PROGRAM MAIN
VAR
	previousTime: ULINT := 0;
	currentTime: ULINT := 0;
	
	loTime: ULINT := 0;
	hiTime: ULINT := 0;
	getTime: GETSYSTEMTIME;
	
	deltaTime: REAL := 0.0;
	
	skogestadPID: Skogestad;
	parallelPID: ParallelPID;

	
	lastPID: REAL := 0;
	useSkogestad: BOOL := TRUE;
	
	init: BOOL := TRUE;
END_VAR

IF init THEN
	lastPID := GVL.kp + GVL.ki + GVL.kd;
	init := FALSE;
END_IF

// Update the useSkogestad flag based if the tuner has changed PID
IF NOT (lastPID = GVL.kp + GVL.ki + GVL.kd) THEN
    useSkogestad := FALSE;
END_IF

// Get the current system time
getTime(timeLoDW => loTime, 
		timeHiDW => hiTime);
currentTime := SHL(hiTime, 32) + loTime;

// Calculate deltaTime
IF (previousTime = 0) THEN
    previousTime := currentTime;
ELSE
    deltaTime := ULINT_TO_REAL(currentTime - previousTime) / 10000000;
    previousTime := currentTime;
END_IF

// Execute the appropriate PID controller
IF NOT (deltaTime = 0.0) THEN
    IF useSkogestad THEN
        skogestadPID(
            rFeedbackVariable := GVL.rTempSensor,
            rSetpoint := GVL.rSetpoint,
            rDeltaTime := deltaTime,
            iOutput => GVL.iHeaterActuator
        );
    ELSE
        parallelPID(
            rFeedbackVariable := GVL.rTempSensor,
            rSetpoint := GVL.rSetpoint,
            rDeltaTime := deltaTime,
            iOutput => GVL.iHeaterActuator
        );
    END_IF
END_IF

END_PROGRAM

(* stored: Version 1.1.0.1, ProductVersion 3.1.4024.12
   POU MAIN: Id {a76c3da7-8f6e-458f-9e74-7b7fc4cfb652}, SpecialFunc None *)
